(* CoDeSys 2.3.9.50 project: 3A.pr6 *)
(* Libraries: STANDARD.LB6 5.6.98 12:03:02 *)

(* POU MAIN, LD *)
PROGRAM MAIN
VAR
	A AT %IX0.0: BOOL;
	Light AT %QX0.0: BOOL;
	t2: TON;
	t1: TON;
END_VAR
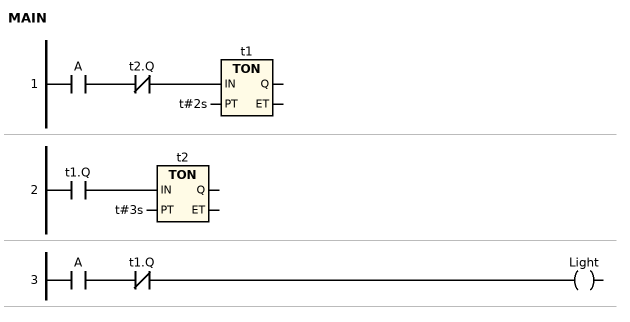
_LD_ (* Ladder Diagram *)
NETWORK 1
	[A] - [/t2.Q] - t1:TON(IN: *, PT: t#2s)
NETWORK 2
	[t1.Q] - t2:TON(IN: *, PT: t#3s)
NETWORK 3
	[A] - [/t1.Q] --- (Light)
_END_LD_
(* the same logic as Structured Text *)
(* Network 1 *)
t1(IN := A AND NOT t2.Q, PT := t#2s);
(* Network 2 *)
t2(IN := t1.Q, PT := t#3s);
(* Network 3 *)
Light := A AND NOT t1.Q;
END_PROGRAM
